FUNCTION_BLOCK EmergencyReactor_2_HMI (* Service Interface Function Block Type *)
  (* Standard: 61499-2 *)
  (* Version 0.0, 7/4/2026, Schneider Electric, template *)
  PACKAGE SE.Nereda;
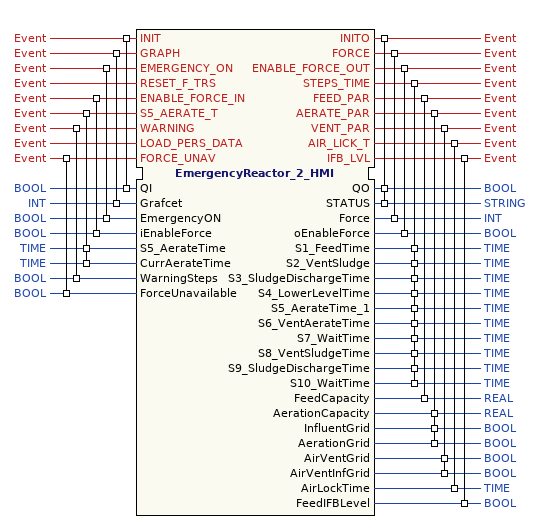
  EVENT_INPUT
    INIT WITH QI;
    GRAPH WITH Grafcet;
    EMERGENCY_ON WITH EmergencyON;
    RESET_F_TRS;
    ENABLE_FORCE_IN WITH iEnableForce;
    S5_AERATE_T WITH S5_AerateTime, CurrAerateTime;
    WARNING WITH WarningSteps;
    LOAD_PERS_DATA;
    FORCE_UNAV WITH ForceUnavailable;
  END_EVENT
  EVENT_OUTPUT
    INITO WITH QO, STATUS;
    FORCE WITH Force;
    ENABLE_FORCE_OUT WITH oEnableForce;
    STEPS_TIME WITH S1_FeedTime, S2_VentSludge, S3_SludgeDischargeTime, S4_LowerLevelTime, S5_AerateTime_1, S6_VentAerateTime, S7_WaitTime, S8_VentSludgeTime, S9_SludgeDischargeTime, S10_WaitTime;
    FEED_PAR WITH FeedCapacity;
    AERATE_PAR WITH AerationCapacity, InfluentGrid, AerationGrid;
    VENT_PAR WITH AirVentGrid, AirVentInfGrid;
    AIR_LICK_T WITH AirLockTime;
    IFB_LVL WITH FeedIFBLevel;
  END_EVENT
  VAR_INPUT
    QI : BOOL;
    Grafcet : INT;
    EmergencyON : BOOL;
    iEnableForce : BOOL;
    S5_AerateTime : TIME;
    CurrAerateTime : TIME;
    WarningSteps : BOOL;
    ForceUnavailable : BOOL;
  END_VAR
  VAR_OUTPUT
    QO : BOOL; (* Event Output Qualifier *)
    STATUS : STRING; (* Service Status *)
    Force : INT;
    oEnableForce : BOOL;
    S1_FeedTime : TIME;
    S2_VentSludge : TIME;
    S3_SludgeDischargeTime : TIME;
    S4_LowerLevelTime : TIME;
    S5_AerateTime_1 : TIME;
    S6_VentAerateTime : TIME;
    S7_WaitTime : TIME;
    S8_VentSludgeTime : TIME;
    S9_SludgeDischargeTime : TIME;
    S10_WaitTime : TIME;
    FeedCapacity : REAL;
    AerationCapacity : REAL;
    InfluentGrid : BOOL;
    AerationGrid : BOOL;
    AirVentGrid : BOOL;
    AirVentInfGrid : BOOL;
    AirLockTime : TIME;
    FeedIFBLevel : BOOL;
  END_VAR
  SERVICE /
    SEQUENCE 
    END_SEQUENCE
  END_SERVICE
END_FUNCTION_BLOCK
